// TIA Portal V17 export
// export: Created 2025-03-07T09:19:50.399801Z, ExportSetting WithDefaults, DisplayName Totally Integrated Automation Portal, DisplayVersion V17 Update 8, DisplayName TIA Portal Openness, DisplayVersion V17 Update 8, DisplayName TIA Portal Version Control Interface, DisplayVersion V17, DisplayName SINAMICS Startdrive Advanced, DisplayVersion V17 SP2, DisplayName SINAMICS Startdrive G110M, G120, G120C, G120D, G120P, G115D, DisplayVersion V17 SP2, DisplayName SINAMICS Startdrive G130, G150, S120, S150, SINAMICS MV, S210, DisplayVersion V17 SP2, DisplayName STEP 7 Professional, DisplayVersion V17 Update 8, DisplayName SINUMERIK ONE STEP 7 Toolbox, DisplayVersion V17 Update 12, DisplayName SINUMERIK 840D sl STEP 7 Toolbox, DisplayVersion V17 Update 12, DisplayName STEP 7 Safety, DisplayVersion V17 Update 6, DisplayName WinCC Advanced, DisplayVersion V17 Update 8
TYPE "CYL_ALARMS_OPN_CLS"
// stored: IsFailsafeCompliant false
   STRUCT
      CLOSED_SIMULTANEITY_1_ALARM : Bool;   // CLOSED SIMULTANEITY 1 ALARM
      CLOSED_TIME_EXCEEDED_1_ALARM : Bool;   // CLOSED TIME EXCEEDED 1 ALARM
      CLOSED_MISSING_1_ALARM : Bool;   // CLOSED MISSING 1 ALARM
      SPARE_1 : Bool;
      CLOSED_SIMULTANEITY_2_ALARM : Bool;   // CLOSED SIMULTANEITY 2 ALARM
      CLOSED_TIME_EXCEEDED_2_ALARM : Bool;   // CLOSED TIME EXCEEDED 2 ALARM
      CLOSED_MISSING_2_ALARM : Bool;   // CLOSED MISSING 2 ALARM
      SPARE_2 : Bool;
      CLOSED_SIMULTANEITY_3_ALARM : Bool;   // CLOSED SIMULTANEITY 3 ALARM
      CLOSED_TIME_EXCEEDED_3_ALARM : Bool;   // CLOSED TIME EXCEEDED 3 ALARM
      CLOSED_MISSING_3_ALARM : Bool;   // CLOSED MISSING 3 ALARM
      SPARE_3 : Bool;
      CLOSED_SIMULTANEITY_4_ALARM : Bool;   // CLOSED SIMULTANEITY 4 ALARM
      CLOSED_TIME_EXCEEDED_4_ALARM : Bool;   // CLOSED TIME EXCEEDED 4 ALARM
      CLOSED_MISSING_4_ALARM : Bool;   // CLOSED MISSING 4 ALARM
      SPARE_4 : Bool;
      CLOSED_OUTPUT_COMMAND_MISSING_ALARM : Bool;   // CLOSED OUTPUT COMMAND MISSING ALARM
      CLOSED_PRESSURE_TIME_EXCEEDED_1_ALARM : Bool;   // CLOSED PRESSURE TIME EXCEEDED 1 ALARM
      CLOSED_PRESSURE_SWITCH_1_ALARM : Bool;   // CLOSED PRESSURE SWITCH 1 ALARM
      CLOSED_PRESSURE_MISSING_1_ALARM : Bool;   // CLOSED PRESSURE MISSING 1 ALARM
      SPARE_5 : Bool;
      CLOSED_PRESSURE_TIME_EXCEEDED_2_ALARM : Bool;   // CLOSED PRESSURE TIME EXCEEDED 2 ALARM
      CLOSED_PRESSURE_SWITCH_2_ALARM : Bool;   // CLOSED PRESSURE SWITCH 2 ALARM
      CLOSED_PRESSURE_MISSING_2_ALARM : Bool;   // CLOSED PRESSURE MISSING 2 ALARM
      SPARE_6 : Bool;
      SPARE_7 : Bool;
      SPARE_8 : Bool;
      SPARE_9 : Bool;
      SPARE_10 : Bool;
      SPARE_11 : Bool;
      SPARE_12 : Bool;
      SPARE_13 : Bool;
      CLOSED_LOW_PRESSURE_TIME_EXCEEDED_ALARM : Bool;   // CLOSED LOW PRESSURE TIME EXCEEDED ALARM
      CLOSED_LOW_PRESSURE_SWITCH_ALARM : Bool;   // CLOSED LOW PRESSURE SWITCH ALARM
      CLOSED_LOW_PRESSURE_MISSING_ALARM : Bool;   // CLOSED LOW PRESSURE MISSING ALARM
      CLOSED_LOW_PRESSURE_OUTPUT_COMMAND_MISSING_ALARM : Bool;   // CLOSED LOW PRESSURE OUTPUT COMMAND MISSING ALARM
      SPARE_15 : Bool;
      SPARE_16 : Bool;
      SPARE_17 : Bool;
      SPARE_18 : Bool;
      OPEN_LOW_PRESSURE_TIME_EXCEEDED_ALARM : Bool;   // OPEN LOW PRESSURE TIME EXCEEDED ALARM
      OPEN_LOW_PRESSURE_SWITCH_ALARM : Bool;   // OPEN LOW PRESSURE SWITCH ALARM
      OPEN_LOW_PRESSURE_MISSING_ALARM : Bool;   // OPEN LOW PRESSURE MISSING ALARM
      OPEN_LOW_PRESSURE_OUTPUT_COMMAND_MISSING_ALARM : Bool;   // OPEN LOW PRESSURE OUTPUT COMMAND MISSING ALARM
      SPARE_23 : Bool;
      SPARE_24 : Bool;
      SPARE_25 : Bool;
      SPARE_26 : Bool;
      OPEN_SIMULTANEITY_1_ALARM : Bool;   // OPEN SIMULTANEITY 1 ALARM
      OPEN_TIME_EXCEEDED_1_ALARM : Bool;   // OPEN TIME EXCEEDED 1 ALARM
      OPEN_MISSING_1_ALARM : Bool;   // OPEN MISSING 1 ALARM
      SPARE_27 : Bool;
      OPEN_SIMULTANEITY_2_ALARM : Bool;   // OPEN SIMULTANEITY 2 ALARM
      OPEN_TIME_EXCEEDED_2_ALARM : Bool;   // OPEN TIME EXCEEDED 2 ALARM
      OPEN_MISSING_2_ALARM : Bool;   // OPEN MISSING 2 ALARM
      SPARE_28 : Bool;
      OPEN_SIMULTANEITY_3_ALARM : Bool;   // OPEN SIMULTANEITY 3 ALARM
      OPEN_TIME_EXCEEDED_3_ALARM : Bool;   // OPEN TIME EXCEEDED 3 ALARM
      OPEN_MISSING_3_ALARM : Bool;   // OPEN MISSING 3 ALARM
      SPARE_29 : Bool;
      OPEN_SIMULTANEITY_4_ALARM : Bool;   // OPEN SIMULTANEITY 4 ALARM
      OPEN_TIME_EXCEEDED_4_ALARM : Bool;   // OPEN TIME EXCEEDED 4 ALARM
      OPEN_MISSING_4_ALARM : Bool;   // OPEN MISSING 4 ALARM
      SPARE_30 : Bool;
      OPEN_OUTPUT_COMMAND_MISSING_ALARM : Bool;   // OPEN OUTPUT COMMAND MISSING ALARM
      OPEN_PRESSURE_TIME_EXCEEDED_1_ALARM : Bool;   // OPEN PRESSURE TIME EXCEEDED 1 ALARM
      OPEN_PRESSURE_SWITCH_1_ALARM : Bool;   // OPEN PRESSURE SWITCH 1 ALARM
      OPEN_PRESSURE_MISSING_1_ALARM : Bool;   // OPEN PRESSURE MISSING 1 ALARM
      SPARE_31 : Bool;
      OPEN_PRESSURE_TIME_EXCEEDED_2_ALARM : Bool;   // OPEN PRESSURE TIME EXCEEDED 2 ALARM
      OPEN_PRESSURE_SWITCH_2_ALARM : Bool;   // OPEN PRESSURE SWITCH 2 ALARM
      OPEN_PRESSURE_MISSING_2_ALARM : Bool;   // OPEN PRESSURE MISSING 2 ALARM
      SPARE_32 : Bool;
      SPARE_33 : Bool;
      SPARE_34 : Bool;
      SPARE_35 : Bool;
      SPARE_36 : Bool;
      SPARE_37 : Bool;
      SPARE_38 : Bool;
      SPARE_39 : Bool;
   END_STRUCT;
END_TYPE
